Fanuc KAREL source: kf00104.KL

-- PROVISIONAL review KL for V940-1; original PC SHA256 8ee2068769aa227ee13452b5eaed3bf1a7d252ca81e87c1c922ffb762093e9a1
-- Incomplete behavior may be omitted. Consult companion uncertainty JSON. Do not deploy.
PROGRAM KF00104
%NOLOCKGROUP
BEGIN
  -- V9_ZERO_TABLE_METADATA_HINT layout=0002_ascii; no indexed target words; source/name/runtime held
  -- UNRESOLVED_PC offsets 5-16; opcodes 2E,23
  -- UNRESOLVED_PC offsets 21-32; opcodes 2E,23
  -- UNRESOLVED_PC offsets 37-57; opcodes 27,27,9D,22,2A,22,31
  -- UNRESOLVED_PC offsets 62-66; opcodes 7F
END KF00104
